// TwinCAT 3 PLC project Oefening1
// ProgramVersion: 3.1.4023.0
// libraries:
//   Tc2_Standard, * (Beckhoff Automation GmbH)
//   Tc2_System, * (Beckhoff Automation GmbH)
//   Tc3_Module, * (Beckhoff Automation GmbH)
// project tree:
//   / GlobalTextList.TcGTLO, PlcTask.TcTTO, Visualization Manager.TcVMO (not stored)
//   POUs/ FB_Knipperlicht.TcPOU, MAIN.TcPOU
//   VISUs/ Oefening1_VISU.TcVIS
// real-time tasks:
//   TASK PlcTask: cycle T#10ms, priority 20, ADS port 350
//   TASK PlcTask1: cycle T#10ms, priority 21, ADS port 351
//   TASK PlcTask2: cycle T#10ms, priority 22, ADS port 352
//   TASK PlcTask3: cycle T#10ms, priority 23, ADS port 353
//   TASK PlcTask4: cycle T#10ms, priority 24, ADS port 354
//   TASK PlcTask5: cycle T#10ms, priority 25, ADS port 355

CONFIGURATION Oefening1
    RESOURCE PLC ON TwinCAT3
        TASK PlcTask(INTERVAL := T#10ms, PRIORITY := 20);
        PROGRAM MAIN WITH PlcTask : MAIN;
    END_RESOURCE
END_CONFIGURATION

// ---- POUs/MAIN.TcPOU
PROGRAM MAIN
VAR
	Knipperlicht: FB_Knipperlicht;
END_VAR

VAR_OUTPUT
	LED : BOOL;
END_VAR

Knipperlicht(
	Enable:= TRUE, 
	OnTime:= T#500MS, 
	OfTime:= T#500MS, 
	Q=> LED);

END_PROGRAM

// ---- POUs/FB_Knipperlicht.TcPOU
FUNCTION_BLOCK FB_Knipperlicht
VAR_INPUT
	Enable : BOOL;	(* activatie knipperlicht*)
	OnTime : TIME;  (* tijd dat de lamp aan is *)
	OfTime : TIME;  (* tijd dat de lamp uit is *)
	CyclesReset : BOOL;
END_VAR

VAR_OUTPUT
	Q: BOOL;		(* het knipperlicht *)
	Freq: REAL;		(* de knipperfrequentie *)
	Duty: REAL;     (* de verhouding aan/totale-tijd *)
	Cycles: REAL;	(* Hoeveelheid cycles voltooid *)
END_VAR

VAR
	Counter : BOOL;
	R_TRIG : R_TRIG;
	tOnTime: TOF;
	tOfTime: TON;
	tTotalTime: TIME; 
END_VAR

IF Enable THEN
	tTotalTime := OnTime + OfTime;
	Duty := (TIME_TO_REAL(OnTime)/(TIME_TO_REAL(OnTime)+TIME_TO_REAL(OfTime))*100);
	Freq := 1000 / (TIME_TO_REAL(OnTime)+TIME_TO_REAL(OfTime));
	
	IF NOT(TIME_TO_REAL(OnTime + OfTime) = 0) THEN
		tOnTime(IN:= NOT tOfTime.Q  , PT:= OnTime, Q=>Q);
		tOfTime(IN:= tOntime.Q 	    , PT:= OfTime, Q=>Q);
	END_IF
	
	R_TRIG(CLK:= Q, Q=> Counter);
	Cycles := Cycles + BOOL_TO_REAL(Counter);
	IF CyclesReset THEN
		Cycles := 0;
	END_IF
ELSE
	Q := FALSE;
END_IF

END_FUNCTION_BLOCK

// ---- VISUs/Oefening1_VISU.TcVIS
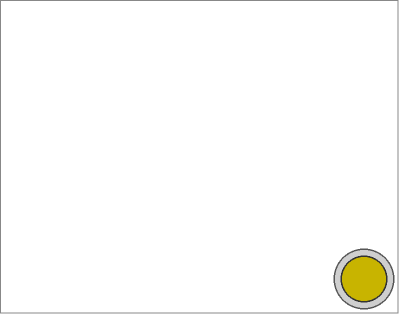
VISUALIZATION Oefening1_VISU  // 399x314
    Lamp1 (329,244 70x70), variable: MAIN.LED, style: Lamp-Lamp1-Yellow
END_VISUALIZATION
